// TIA Portal V16 export
// export: Created 2021-11-15T21:16:57.6885547Z, ExportSetting WithDefaults, WithReadOnly, DisplayName Totally Integrated Automation Portal, DisplayVersion V16 Update 3, DisplayName TIA Portal Version Control Interface, DisplayVersion V16 Update 2, DisplayName TIA Portal Openness, DisplayVersion V16 Update 3, DisplayName SINAMICS Startdrive Advanced, DisplayVersion V16, DisplayName SINAMICS Startdrive G130, G150, S120, S150, SINAMICS MV, S210, DisplayVersion V16, DisplayName SINAMICS Startdrive G110M, G120, G120C, G120D, G120P, DisplayVersion V16, DisplayName STEP 7 Professional, DisplayVersion V16 Update 3, DisplayName SIMATIC Energy Suite, DisplayVersion V16, DisplayName STEP 7 Safety, DisplayVersion V16, DisplayName WinCC Advanced, DisplayVersion V16 Update 3
FUNCTION "Export" : Void   // FC2, LAD
{ S7_Optimized_Access := 'TRUE' }
VERSION : 0.1
// stored: AutoNumber true, CodeModifiedDate 2021-11-15T21:14:45.9278125Z, CompileDate 2021-11-15T21:14:56.9551563Z, CreationDate 2021-11-15T21:12:04.4639454Z, HandleErrorsWithinBlock false, InterfaceModifiedDate 2021-11-15T21:12:04.4639454Z, IsConsistent true, IsIECCheckEnabled false, IsKnowHowProtected false, IsWriteProtected false, LibraryConformanceStatus Avviso: Il blocco contiene accessi diretti a ingressi, uscite, merker, accessi indiretti a registri o accessi indiretti ad aree di memoria esterne sconosciute al momento della compilazione., ModifiedDate 2021-11-15T21:14:45.9278125Z, ParameterModified 2021-11-15T21:12:04.4639454Z, PLCSimAdvancedSupport true, SetENOAutomatically false, StructureModified 2021-11-15T21:12:04.4639454Z, UDAEnableTagReadback false
BEGIN

REGION Network 1
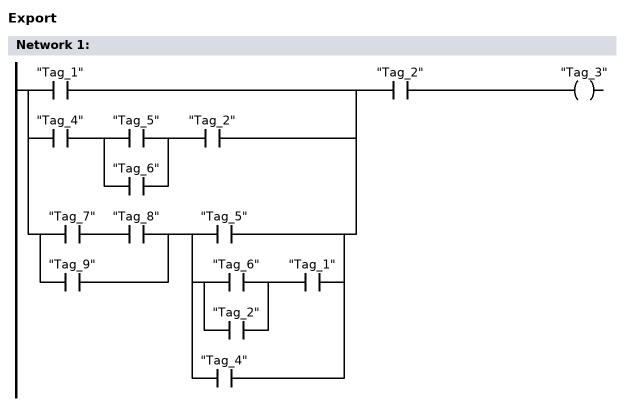
   "Tag_3" := ("Tag_1" OR ("Tag_4" AND ("Tag_5" OR "Tag_6") AND "Tag_2") OR ((("Tag_7" AND "Tag_8") OR "Tag_9") AND ("Tag_5" OR (("Tag_6" OR "Tag_2") AND "Tag_1") OR "Tag_4"))) AND "Tag_2";
END_REGION
END_FUNCTION
